(* PLC project Sin nombre, Desconocido Sin nombre 1 *)
(* stored: creationDateTime 2022-10-17T16:56:25, modificationDateTime 2024-10-31T16:44:36 *)

PROGRAM program0
  VAR
    Out1 AT %QX0.0 : BOOL := 0;
    Sensor AT %IX0.0 : BOOL := 0;
  END_VAR
  VAR
    Inputt : BOOL := 0;
    Inputt0 : BOOL := 0;
    tiempo : INT := 0;
    TP1 : TP;
    CTUD0 : CTUD;
    TP3 : TP;
    TOF2 : TOF;
    CTU1 : CTU;
    TP4 : TP;
    TOF3 : TOF;
    CTU2 : CTU;
    TP5 : TP;
    TOF4 : TOF;
    CTU3 : CTU;
    TP6 : TP;
    TOF5 : TOF;
    CTU4 : CTU;
    TON0 : TON;
    TP0 : TP;
    TP2 : TP;
    TP7 : TP;
  END_VAR
  VAR  (* added by the conversion: wires and edge detectors of the diagram *)
    R_TRIG1 : R_TRIG;
    _INT_TO_BOOL91_OUT : BOOL;
    _NOT92_OUT : BOOL;
    R_TRIG2 : R_TRIG;
    R_TRIG3 : R_TRIG;
    R_TRIG4 : R_TRIG;
    R_TRIG5 : R_TRIG;
    R_TRIG6 : R_TRIG;
  END_VAR

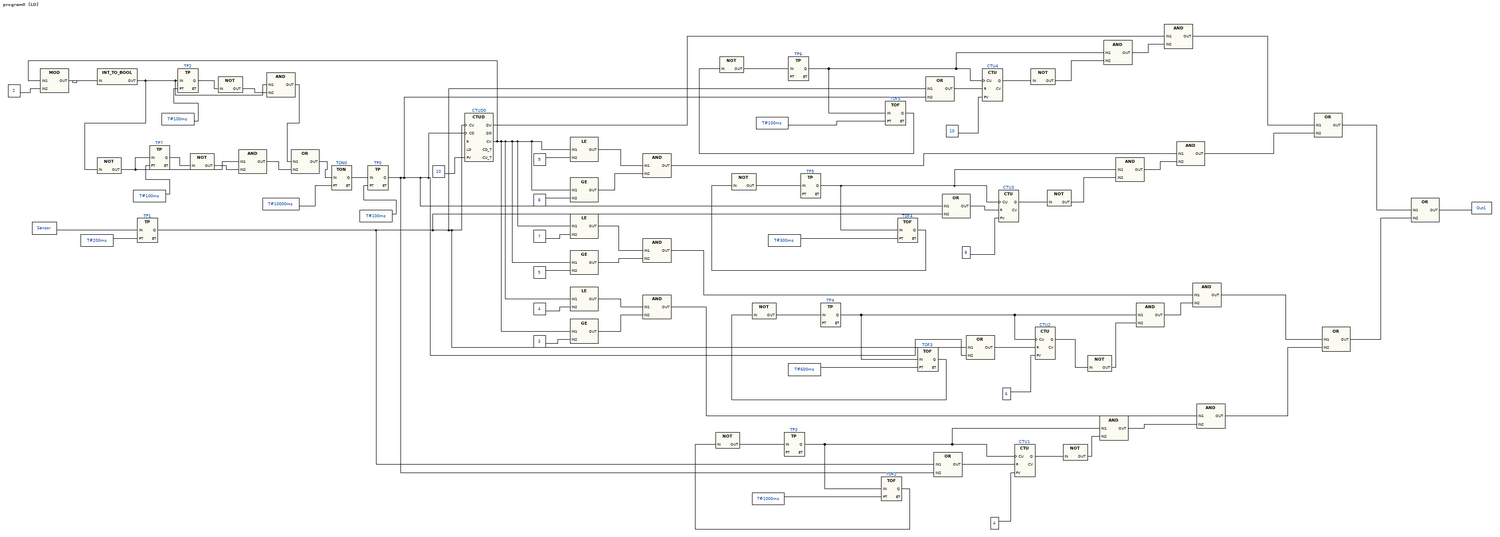
(* LD diagram, written out as Structured Text *)
TP1(IN := Sensor, PT := T#200ms);
R_TRIG1(CLK := TP1.Q);
_INT_TO_BOOL91_OUT := INT_TO_BOOL(CTUD0.CV MOD 2);
TP2(IN := _INT_TO_BOOL91_OUT, PT := T#100ms);
_NOT92_OUT := NOT _INT_TO_BOOL91_OUT;
TP7(IN := _NOT92_OUT, PT := T#100ms);
TON0(IN := _INT_TO_BOOL91_OUT AND NOT TP2.Q OR _NOT92_OUT AND NOT TP7.Q, PT := T#10000ms);
TP0(IN := TON0.Q, PT := T#100ms);
R_TRIG2(CLK := TP0.Q);
CTUD0(CU := R_TRIG1.Q, CD := R_TRIG2.Q, PV := 10);
TOF5(IN := TP6.Q, PT := T#100ms);
TP6(IN := NOT TOF5.Q);
R_TRIG3(CLK := TP6.Q);
CTU4(CU := R_TRIG3.Q, R := TP1.Q OR TP0.Q, PV := 10);
TOF4(IN := TP5.Q, PT := T#300ms);
TP5(IN := NOT TOF4.Q);
R_TRIG4(CLK := TP5.Q);
CTU3(CU := R_TRIG4.Q, R := TP0.Q OR TP1.Q, PV := 8);
TOF3(IN := TP4.Q, PT := T#600ms);
TP4(IN := NOT TOF3.Q);
R_TRIG5(CLK := TP4.Q);
CTU2(CU := R_TRIG5.Q, R := TP1.Q OR TP0.Q, PV := 6);
TOF2(IN := TP3.Q, PT := T#1000ms);
TP3(IN := NOT TOF2.Q);
R_TRIG6(CLK := TP3.Q);
CTU1(CU := R_TRIG6.Q, R := TP1.Q OR TP0.Q, PV := 4);
Out1 := CTUD0.QU AND TP6.Q AND NOT CTU4.Q OR CTUD0.CV <= 9 AND CTUD0.CV >= 8 AND TP5.Q AND NOT CTU3.Q OR CTUD0.CV <= 7 AND CTUD0.CV >= 5 AND TP4.Q AND NOT CTU2.Q OR CTUD0.CV <= 4 AND CTUD0.CV >= 3 AND TP3.Q AND NOT CTU1.Q;
END_PROGRAM

CONFIGURATION Config0
  RESOURCE Res0 ON PLC
    TASK task0(INTERVAL := T#20ms, PRIORITY := 0);
    PROGRAM instance0 WITH task0 : program0;
  END_RESOURCE
END_CONFIGURATION
